FUNCTION F_DeviceTwin_GetReportedProperties : STRING(2000)
VAR_INPUT
END_VAR
VAR
	(* JSON document *)
	fbJsonDeviceInfo 	: FB_JsonSaxWriter;
	sJsonDocDeviceInfo 	: STRING(2000);
END_VAR

fbJsonDeviceInfo.StartObject();
fbJsonDeviceInfo.AddKey('Device');
fbJsonDeviceInfo.StartObject();
fbJsonDeviceInfo.AddKey('Location');
fbJsonDeviceInfo.StartObject();
fbJsonDeviceInfo.AddKey('Latitude');
fbJsonDeviceInfo.AddString('51.881034');
fbJsonDeviceInfo.AddKey('Longitude');
fbJsonDeviceInfo.AddString('8.491037');
fbJsonDeviceInfo.EndObject();
fbJsonDeviceInfo.EndObject();
fbJsonDeviceInfo.AddKey('System');
fbJsonDeviceInfo.StartObject();
fbJsonDeviceInfo.AddKey('Manufacturer');
fbJsonDeviceInfo.AddString('Beckhoff Automation');
fbJsonDeviceInfo.AddKey('Firmware');
fbJsonDeviceInfo.AddString('1.42');
fbJsonDeviceInfo.AddKey('InstalledRAM');
fbJsonDeviceInfo.AddString('4 GB');
fbJsonDeviceInfo.AddKey('Processor');
fbJsonDeviceInfo.AddString('Intel Core i5');
fbJsonDeviceInfo.EndObject();
fbJsonDeviceInfo.EndObject();
sJsonDocDeviceInfo := fbJsonDeviceInfo.GetDocument();
F_DeviceTwin_GetReportedProperties := sJsonDocDeviceInfo;

END_FUNCTION

(* stored: Version 1.1.0.1, ProductVersion 3.1.4022.3
   POU F_DeviceTwin_GetReportedProperties: Id {a53f3d7c-92da-4596-84cb-b86a0f97ef79}, SpecialFunc None *)
